(*
SPDX-FileCopyrightText: © 2026 Oleksandr Tiutyk <trofimich@gmail.com>
SPDX-License-Identifier: MIT
License: https://opensource.org/license/mit
*)

INTERFACE IDataMemberOutOfRangeException EXTENDS IGeneralException

METHOD Throw
VAR_INPUT
	sourceNamespaceName : STRING;
	sourceClassName : STRING;
	sourcePOUName : STRING;
	sourcePosition : STRING;
	dataMemberName : STRING;
	dataMemberValue : ANY;
END_VAR
END_METHOD

END_INTERFACE

(* stored: Version 1.1.0.1
   Itf IDataMemberOutOfRangeException: Id {cf663f39-5e05-4307-91b0-0444aac88c2e}
   Method Throw: Id {c468a2b6-6032-48d2-a9d4-533017cb99d6} *)
